{attribute 'qualified_only'}
{attribute 'strict'}
TYPE E_CtrlState :
(
	STOPPED 	:= 0,
	IDLE		:= 1,
	RUNNING		:= 2,
	STOPPING	:= 3
);
END_TYPE

(* stored: Version 1.1.0.1, ProductVersion 3.1.4024.12
   DUT E_CtrlState: Id {4520cd68-e4e5-494a-a3f4-7735f77a3455} *)
